PROGRAM TEST_MAIN
VAR
  test_event: TestEvent;
  test_ads_logger: TestADSLogger;
  test_csv_logger: TestCSVLogger;
  test_utils: TestUtils;
END_VAR

TcUnit.RUN();

END_PROGRAM

(* stored: Version 1.1.0.1, ProductVersion 3.1.4024.9
   POU TEST_MAIN: Id {e0fe771e-7548-4546-bb6c-2059f20a9739}, SpecialFunc None *)
